TYPE ST_MESSAGE_STATE :
STRUCT
  State         : E_MESSAGE_STATE;  // as always... combined value of Cmd equivalent and e_progress
END_STRUCT
END_TYPE

(* stored: Version 1.1.0.1, ProductVersion 3.1.4026.20
   DUT ST_MESSAGE_STATE: Id {105d3d6a-2716-411a-add9-5cb1c7beaf43} *)
